ABB RAPID module: Wobj_wobj_C1.mod

MODULE Wobj_wobj_C1
	! Points are read in order of declaration.
  ! Please do not change the order of points!

  LOCAL PERS robtarget pWobj_U_PointX1:=[[-1279.58,-2151.72,-615.7369],[0.00633935770019889,-0.720863401889801,0.693027794361115,-0.00531704723834991],[-2,0,1,0],[0,9E+09,9E+09,9E+09,9E+09,9E+09]];
	LOCAL PERS robtarget pWobj_U_PointX2:=[[-763.1923,-2127.489,-615.7349],[0.00634018890559673,-0.720860481262207,0.693030774593353,-0.00531714595854282],[-2,0,1,0],[0,9E+09,9E+09,9E+09,9E+09,9E+09]];
	LOCAL PERS robtarget pWobj_U_PointY1:=[[-1309.352,-1528.973,-614.7366],[0.00633547129109502,-0.720859944820404,0.693031430244446,-0.00531624583527446],[-2,0,1,0],[0,9E+09,9E+09,9E+09,9E+09,9E+09]];

ENDMODULE
